// TIA Portal V19 export
FUNCTION_BLOCK "DecoilersHU_FB"   // FB28, LAD
// stored: MemoryReserve 100, SetENOAutomatically false
   VAR_INPUT
      AreaInterface : "AreaInterface";
      ZSI : "udt_ZoneSafetyInterface";
      DSI : "udt_DeviceSafetyInterface";
      DataIn : Struct
         Pb_Stop : Bool;
         Pb_Start : Bool;
      END_STRUCT;
      CIn : Struct
         EnableStopStopDueDoorOpeningRequest : Bool := TRUE;
         EnableStopInPhase : Bool;
         EnableStopProgrammed : Bool;
         PressureReq : Bool;
      END_STRUCT;
   END_VAR
   VAR_OUTPUT
      MachineInterface : "MachineInterface";
      DataOut : Struct
         Pressure_V : Bool;
      END_STRUCT;
      COut : Struct
         Standstill : Bool;
         Run_CheckNext : Bool;
         CtrlSafe : Bool;
         PressureRunning : Bool;
      END_STRUCT;
   END_VAR
   VAR
      Sts : Struct
         Standstill : Bool;
         AlarmsPresence : Bool;
         WarningsPresence : Bool;
         Cnd : Bool;
      END_STRUCT;
      Ctrl : Struct
         StopDueDoorOpeningRequest : Bool;
         StopInPhase : Bool;
         StopProgrammed : Bool;
         StopAborting : Bool;
         Run : Bool;
         Run_Man : Bool;
         Run_Aut : Bool;
      END_STRUCT;
      Alarm : Struct
         Pump : "MotorAlr";
      END_STRUCT;
      Warning : Struct
         NotAutReady : Bool;
      END_STRUCT;
      Pump_M : "Motor";
      TON_NoPendingCmd : IEC_TIMER;
      TON_Inactivity : IEC_TIMER;
      TON_Pressure { S7_SetPoint := 'True'} : IEC_TIMER;
      Aux : Struct
         Pb_Start : Bool;
      END_STRUCT;
   END_VAR
   VAR_TEMP   // added for the SCL form of the ladder/FBD networks
      _w1 : Bool;
   END_VAR
BEGIN

REGION Network 1: <<< MACHINE STOP >>>
END_REGION

REGION Network 2: Stop due next door opening
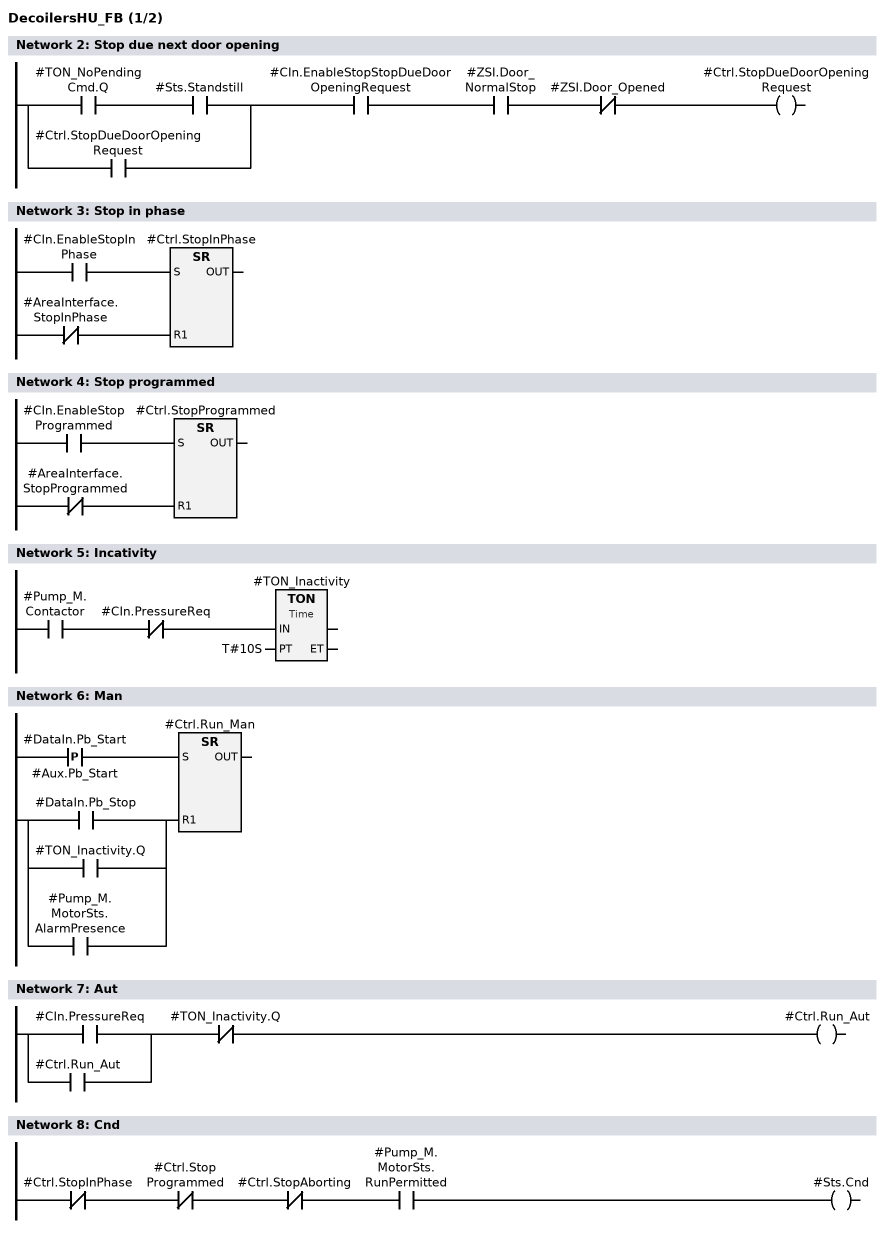
   RUNG wire#powerrail
      Contact( #TON_NoPendingCmd.Q )
      Contact( #Sts.Standstill )
      wire#w1
      Contact( #CIn.EnableStopStopDueDoorOpeningRequest )
      Contact( #ZSI.Door_NormalStop )
      I_Contact( #ZSI.Door_Opened )
      Coil( #Ctrl.StopDueDoorOpeningRequest )
   END_RUNG
   RUNG wire#powerrail
      Contact( #Ctrl.StopDueDoorOpeningRequest )
   END_RUNG wire#w1
   // the same network as SCL:
   #Ctrl.StopDueDoorOpeningRequest := ((#TON_NoPendingCmd.Q AND #Sts.Standstill) OR #Ctrl.StopDueDoorOpeningRequest) AND #CIn.EnableStopStopDueDoorOpeningRequest AND #ZSI.Door_NormalStop AND NOT #ZSI.Door_Opened;
END_REGION

REGION Network 3: Stop in phase
   RUNG wire#powerrail
      Contact( #CIn.EnableStopInPhase )
      S_SR(operand := #Ctrl.StopInPhase, r1 := wire#w1)
   END_RUNG
   RUNG wire#powerrail
      I_Contact( #AreaInterface.StopInPhase )
   END_RUNG wire#w1
   // the same network as SCL:
   IF #CIn.EnableStopInPhase THEN
       #Ctrl.StopInPhase := TRUE;   // SR flip-flop
   END_IF;
   IF NOT #AreaInterface.StopInPhase THEN #Ctrl.StopInPhase := FALSE; END_IF;
END_REGION

REGION Network 4: Stop programmed
   RUNG wire#powerrail
      Contact( #CIn.EnableStopProgrammed )
      S_SR(operand := #Ctrl.StopProgrammed, r1 := wire#w1)
   END_RUNG
   RUNG wire#powerrail
      I_Contact( #AreaInterface.StopProgrammed )
   END_RUNG wire#w1
   // the same network as SCL:
   IF #CIn.EnableStopProgrammed THEN
       #Ctrl.StopProgrammed := TRUE;   // SR flip-flop
   END_IF;
   IF NOT #AreaInterface.StopProgrammed THEN #Ctrl.StopProgrammed := FALSE; END_IF;
END_REGION

REGION Network 5: Incativity
   RUNG wire#powerrail
      Contact( #Pump_M.Contactor )
      I_Contact( #CIn.PressureReq )
      { S7_Templates := "time_type := Time" } #TON_Inactivity.TON(pt := T#10S, et =>)
   END_RUNG
   // the same network as SCL:
   #TON_Inactivity.TON(IN := #Pump_M.Contactor AND NOT #CIn.PressureReq, PT := T#10S);
END_REGION

REGION Network 6: Man
   RUNG wire#powerrail
      P_Contact(operand := #DataIn.Pb_Start, bit := #Aux.Pb_Start)
      S_SR(operand := #Ctrl.Run_Man, r1 := wire#w1)
   END_RUNG
   RUNG wire#powerrail
      Contact( #DataIn.Pb_Stop )
   END_RUNG wire#w1
   RUNG wire#powerrail
      Contact( #TON_Inactivity.Q )
   END_RUNG wire#w1
   RUNG wire#powerrail
      Contact( #Pump_M.MotorSts.AlarmPresence )
   END_RUNG wire#w1
   // the same network as SCL:
   #_w1 := #DataIn.Pb_Start AND NOT #Aux.Pb_Start;   // rising edge of #DataIn.Pb_Start
   #Aux.Pb_Start := #DataIn.Pb_Start;
   IF #_w1 THEN
       #Ctrl.Run_Man := TRUE;   // SR flip-flop
   END_IF;
   IF #DataIn.Pb_Stop OR #TON_Inactivity.Q OR #Pump_M.MotorSts.AlarmPresence THEN
       #Ctrl.Run_Man := FALSE;
   END_IF;
END_REGION

REGION Network 7: Aut
   RUNG wire#powerrail
      Contact( #CIn.PressureReq )
      wire#w1
      I_Contact( #TON_Inactivity.Q )
      Coil( #Ctrl.Run_Aut )
   END_RUNG
   RUNG wire#powerrail
      Contact( #Ctrl.Run_Aut )
   END_RUNG wire#w1
   // the same network as SCL:
   #Ctrl.Run_Aut := (#CIn.PressureReq OR #Ctrl.Run_Aut) AND NOT #TON_Inactivity.Q;
END_REGION

REGION Network 8: Cnd
   RUNG wire#powerrail
      I_Contact( #Ctrl.StopInPhase )
      I_Contact( #Ctrl.StopProgrammed )
      I_Contact( #Ctrl.StopAborting )
      Contact( #Pump_M.MotorSts.RunPermitted )
      Coil( #Sts.Cnd )
   END_RUNG
   // the same network as SCL:
   #Sts.Cnd := NOT #Ctrl.StopInPhase AND NOT #Ctrl.StopProgrammed AND NOT #Ctrl.StopAborting AND #Pump_M.MotorSts.RunPermitted;
END_REGION

REGION Network 9: Run command
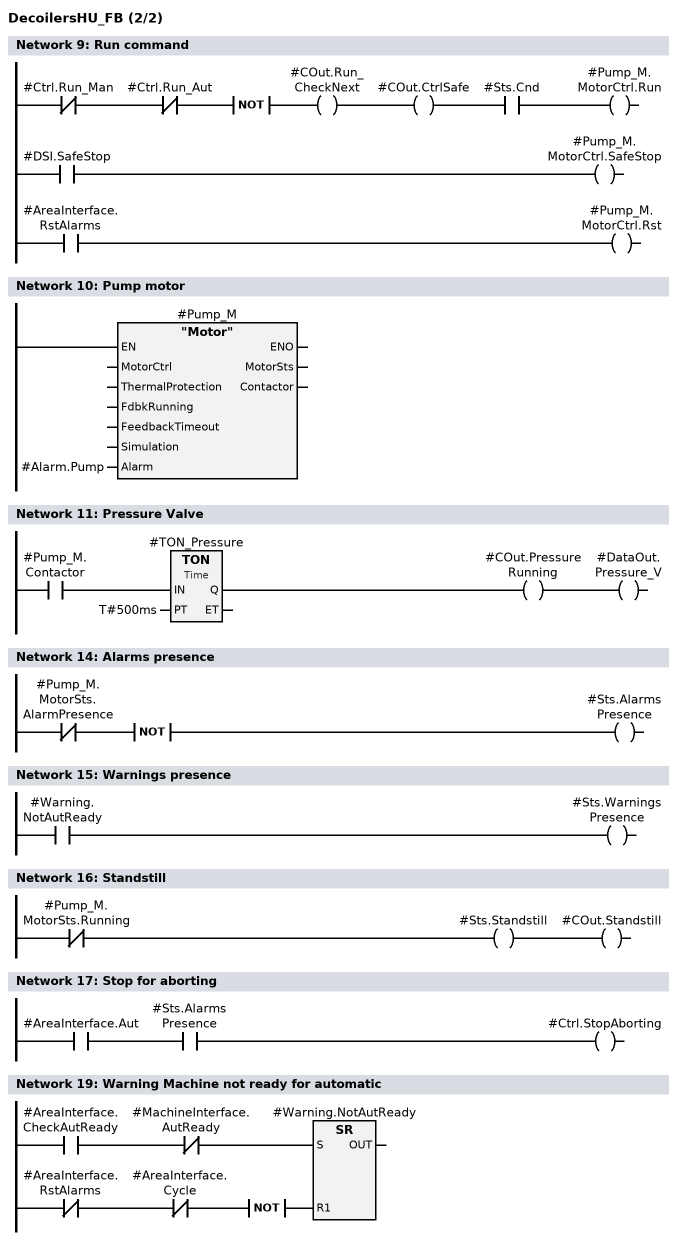
   RUNG wire#powerrail
      I_Contact( #Ctrl.Run_Man )
      I_Contact( #Ctrl.Run_Aut )
      Not()
      Coil( #COut.Run_CheckNext )
      Coil( #COut.CtrlSafe )
      Contact( #Sts.Cnd )
      Coil( #Pump_M.MotorCtrl.Run )
   END_RUNG
   RUNG wire#powerrail
      Contact( #DSI.SafeStop )
      Coil( #Pump_M.MotorCtrl.SafeStop )
   END_RUNG
   RUNG wire#powerrail
      Contact( #AreaInterface.RstAlarms )
      Coil( #Pump_M.MotorCtrl.Rst )
   END_RUNG
   // the same network as SCL:
   #COut.Run_CheckNext := NOT (NOT #Ctrl.Run_Man AND NOT #Ctrl.Run_Aut);
   #COut.CtrlSafe := #COut.Run_CheckNext;
   #Pump_M.MotorCtrl.Run := #COut.Run_CheckNext AND #Sts.Cnd;
   #Pump_M.MotorCtrl.SafeStop := #DSI.SafeStop;
   #Pump_M.MotorCtrl.Rst := #AreaInterface.RstAlarms;
END_REGION

REGION Network 10: Pump motor
   RUNG wire#powerrail
      #Pump_M(MotorCtrl :=, ThermalProtection :=, FdbkRunning :=, FeedbackTimeout :=, Simulation :=, Alarm := #Alarm.Pump, MotorSts =>, Contactor =>)
   END_RUNG
   // the same network as SCL:
   #Pump_M(Alarm := #Alarm.Pump);   // "Motor"
END_REGION

REGION Network 11: Pressure Valve
   RUNG wire#powerrail
      Contact( #Pump_M.Contactor )
      { S7_Templates := "time_type := Time" } #TON_Pressure.TON(pt := T#500ms, et =>)
      Coil( #COut.PressureRunning )
      Coil( #DataOut.Pressure_V )
   END_RUNG
   // the same network as SCL:
   #TON_Pressure.TON(IN := #Pump_M.Contactor, PT := T#500ms);
   #COut.PressureRunning := #TON_Pressure.Q;
   #DataOut.Pressure_V := #TON_Pressure.Q;
END_REGION

REGION Network 12: >
END_REGION

REGION Network 13: <<< MACHINE STATUS >>>
END_REGION

REGION Network 14: Alarms presence
   RUNG wire#powerrail
      I_Contact( #Pump_M.MotorSts.AlarmPresence )
      Not()
      Coil( #Sts.AlarmsPresence )
   END_RUNG
   // the same network as SCL:
   #Sts.AlarmsPresence := NOT (NOT #Pump_M.MotorSts.AlarmPresence);
END_REGION

REGION Network 15: Warnings presence
   RUNG wire#powerrail
      Contact( #Warning.NotAutReady )
      Coil( #Sts.WarningsPresence )
   END_RUNG
   // the same network as SCL:
   #Sts.WarningsPresence := #Warning.NotAutReady;
END_REGION

REGION Network 16: Standstill
   RUNG wire#powerrail
      I_Contact( #Pump_M.MotorSts.Running )
      Coil( #Sts.Standstill )
      Coil( #COut.Standstill )
   END_RUNG
   // the same network as SCL:
   #Sts.Standstill := NOT #Pump_M.MotorSts.Running;
   #COut.Standstill := NOT #Pump_M.MotorSts.Running;
END_REGION

REGION Network 17: Stop for aborting
   RUNG wire#powerrail
      Contact( #AreaInterface.Aut )
      Contact( #Sts.AlarmsPresence )
      Coil( #Ctrl.StopAborting )
   END_RUNG
   // the same network as SCL:
   #Ctrl.StopAborting := #AreaInterface.Aut AND #Sts.AlarmsPresence;
END_REGION

REGION Network 18 (SCL): Collect machine to zone interface

   #MachineInterface.AutReady := #AreaInterface.Aut AND NOT #Sts.AlarmsPresence;
   #MachineInterface.Aborting := #Ctrl.StopAborting;
   #MachineInterface.MotionsStandStill := #TON_NoPendingCmd.Q AND #Sts.Standstill;
   #MachineInterface.AckStopInPhase := #Ctrl.StopInPhase  AND #MachineInterface.MotionsStandStill;
   #MachineInterface.AckStopProgrammed := #Ctrl.StopProgrammed AND #MachineInterface.MotionsStandStill;
   #MachineInterface.AlarmsPresence := #Sts.AlarmsPresence;
   #MachineInterface.WarningPresence := #Sts.WarningsPresence;
END_REGION

REGION Network 19: Warning Machine not ready for automatic
   RUNG wire#powerrail
      Contact( #AreaInterface.CheckAutReady )
      I_Contact( #MachineInterface.AutReady )
      S_SR(operand := #Warning.NotAutReady, r1 := wire#w1)
   END_RUNG
   RUNG wire#powerrail
      I_Contact( #AreaInterface.RstAlarms )
      I_Contact( #AreaInterface.Cycle )
      Not()
   END_RUNG wire#w1
   // the same network as SCL:
   IF #AreaInterface.CheckAutReady AND NOT #MachineInterface.AutReady THEN
       #Warning.NotAutReady := TRUE;   // SR flip-flop
   END_IF;
   IF NOT (NOT #AreaInterface.RstAlarms AND NOT #AreaInterface.Cycle) THEN
       #Warning.NotAutReady := FALSE;
   END_IF;
END_REGION

REGION Network 20: >
END_REGION

REGION Network 21: >
END_REGION

REGION Network 22: >
END_REGION
END_FUNCTION_BLOCK
